SUBAPPLICATION Uebung_039_sub_NumbAnzeig_AX (* Spiegelabfolge V2 mit Schrittkette SUB Num *)
  (* Standard: 61499-2; Description: Copyright (c) 2023 Meisterschulen am Ostbahnhof This program and the accompanying materials are made available under the terms of the Eclipse Public License 2.0 which is available at https://www.eclipse.org/legal/epl-2.0/ SPDX-License-Identifier: EPL-2.0 *)
  (* Version 1.0, 2024-03-03, Franz Höpfinger, Meisterschulen am Ostbahnhof, initial API and implementation and/or initial documentation *)
  PACKAGE Uebungen;
  IMPORT Uebungen::const::UT::DefaultPool::OutputNumber_N1;
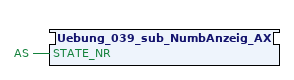
  SOCKETS
    STATE_NR : adapter::types::unidirectional::AS;
  END_SOCKETS
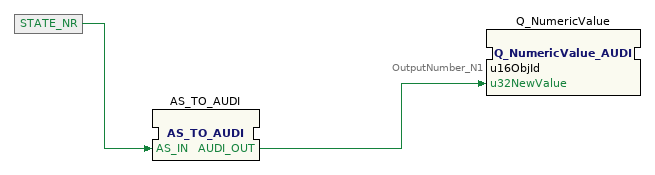
  FBS
    Q_NumericValue : isobus::UT::Q::Q_NumericValue_AUDI(u16ObjId := OutputNumber_N1);
    AS_TO_AUDI : adapter::conversion::unidirectional::AS_TO_AUDI;
  END_FBS
  ADAPTER_CONNECTIONS
    AS_TO_AUDI.AUDI_OUT TO Q_NumericValue.u32NewValue;
    STATE_NR TO AS_TO_AUDI.AS_IN;
  END_CONNECTIONS
END_SUBAPPLICATION
